{attribute 'reflection'}
FUNCTION_BLOCK Object
VAR_OUTPUT 
  busy: BOOL;
	done: BOOL;
  ready: BOOL;
//	error: BOOL;
  error_id: UDINT;
END_VAR
VAR
  {attribute 'instance-path'}
  {attribute 'noinit'}
  fb_id: STRING(255);
END_VAR

END_FUNCTION_BLOCK

(* stored: Version 1.1.0.1, ProductVersion 3.1.4022.18
   POU Object: Id {1e66cee1-d60b-4e6a-8a9b-a522199e7de9}, SpecialFunc None *)
